TYPE _00BE31_HWTOPLC_PDOS :
STRUCT
	
	inputByte_0 	 : BYTE;
	inputByte_1  : BYTE;

END_STRUCT
END_TYPE

(* stored: Version 1.1.0.1
   DUT _00BE31_HWTOPLC_PDOS: Id {f4f4bbe7-f125-4b81-a2bf-53842aac1165} *)
